(* IEC 61131-3 sources: Lasal/CPU_5344_V01/Class/cmServo, 1 file *)

(* ---- cmServo.st ---- *)
(*!
<Class
	Name               = "cmServo"
	Revision           = "1.0"
	RealtimeTask       = "false"
	CyclicTask         = "true"
	DefCyclictime      = "10 ms"
	BackgroundTask     = "true"
	DefBackground      = "500 ms"
	Sigmatek           = "false"
	OSInterface        = "false"
	HighPriority       = "false"
	Automatic          = "false"
	UpdateMode         = "Prescan"
	SharedCommandTable = "true"
	Objectsize         = "(570,2640)">
	<Channels>
		<Server Name="calcReqSpeed" Visualized="false" Initialize="false" WriteProtected="true" Retentive="false"/>
		<Server Name="csPowerOffServo" Visualized="false" Initialize="false" WriteProtected="false" Retentive="false"/>
		<Server Name="firstPos" Visualized="false" Initialize="false" WriteProtected="false" Retentive="false"/>
		<Server Name="parExtraIFactor" Visualized="true" Initialize="true" DefValue="0" WriteProtected="false" Retentive="File"/>
		<Server Name="parHomeAgain" Visualized="true" Initialize="false" WriteProtected="false" Retentive="false"/>
		<Server Name="parIFactor" Visualized="true" Initialize="true" DefValue="0" WriteProtected="false" Retentive="File"/>
		<Server Name="parInPosBand" Visualized="true" Initialize="true" DefValue="100" WriteProtected="false" Retentive="File" Comment="max difference between act real pos and req pos  (*100)&#13;&#10;in thousands of mm for sts.InPos"/>
		<Server Name="parJogTime" Visualized="true" Initialize="true" DefValue="500" WriteProtected="false" Retentive="File"/>
		<Server Name="parKeepControllerOn" Visualized="true" Initialize="true" WriteProtected="false" Retentive="File"/>
		<Server Name="parLastPieceBand" Visualized="true" Initialize="true" DefValue="1000" WriteProtected="false" Retentive="File"/>
		<Server Name="parManualSpeed" Visualized="true" Initialize="true" DefValue="500" WriteProtected="false" Retentive="File"/>
		<Server Name="parMaxAcc" Visualized="true" Initialize="true" DefValue="10000" WriteProtected="false" Retentive="File"/>
		<Server Name="parMaxDec" Visualized="true" Initialize="true" DefValue="10000" WriteProtected="false" Retentive="File"/>
		<Server Name="parMaxPos" Visualized="true" Initialize="true" DefValue="1500000" WriteProtected="false" Retentive="File"/>
		<Server Name="parMaxSpeed" Visualized="true" Initialize="true" DefValue="10000" WriteProtected="false" Retentive="File"/>
		<Server Name="parMinPos" Visualized="true" Initialize="true" DefValue="0" WriteProtected="false" Retentive="File"/>
		<Server Name="parNoRefSwitch" Visualized="true" Initialize="true" WriteProtected="false" Retentive="File"/>
		<Server Name="parOverrideSimulateServo" Visualized="false" Initialize="false" WriteProtected="false" Retentive="File"/>
		<Server Name="parRefDirPositive" Visualized="true" Initialize="true" DefValue="1" WriteProtected="false" Retentive="File"/>
		<Server Name="parRefPos" Visualized="true" Initialize="true" DefValue="1500000" WriteProtected="false" Retentive="File"/>
		<Server Name="parRefSpeed" Visualized="true" Initialize="true" DefValue="1000" WriteProtected="false" Retentive="File"/>
		<Server Name="parTimeBrakeOff" Visualized="true" Initialize="true" DefValue="200" WriteProtected="false" Retentive="File"/>
		<Server Name="parTimeBrakeOn" Visualized="true" Initialize="true" DefValue="200" WriteProtected="false" Retentive="File"/>
		<Server Name="parTimeControllerOn" Visualized="true" Initialize="true" DefValue="100" WriteProtected="false" Retentive="File"/>
		<Server Name="parTimeOutTime" Visualized="true" Initialize="true" DefValue="120000" WriteProtected="false" Retentive="File"/>
		<Server Name="parWaitInPosTime" Visualized="true" Initialize="true" DefValue="100" WriteProtected="false" Retentive="File"/>
		<Server Name="PendelOn" Visualized="false" Initialize="false" WriteProtected="false" Retentive="false"/>
		<Server Name="reqAcc" Visualized="true" Initialize="false" WriteProtected="false" Retentive="false"/>
		<Server Name="reqDec" Visualized="true" Initialize="false" WriteProtected="false" Retentive="false"/>
		<Server Name="reqPos" Visualized="true" Initialize="false" WriteProtected="false" Retentive="false"/>
		<Server Name="reqSpeed" Visualized="true" Initialize="false" WriteProtected="false" Retentive="false"/>
		<Server Name="secondPos" Visualized="false" Initialize="false" WriteProtected="false" Retentive="false"/>
		<Server Name="stsActRealPos" Visualized="true" Initialize="false" WriteProtected="true" Retentive="false"/>
		<Server Name="stsAllSimuActive" Visualized="false" Initialize="false" WriteProtected="true" Retentive="false"/>
		<Server Name="stsControllerIsOn" Visualized="true" Initialize="false" WriteProtected="true" Retentive="false"/>
		<Server Name="stsInPos" Visualized="true" Initialize="false" WriteProtected="true" Retentive="false"/>
		<Server Name="stsIsHomed" Visualized="true" Initialize="false" WriteProtected="false" Retentive="false"/>
		<Server Name="stsPos" Visualized="true" Initialize="false" WriteProtected="true" Retentive="false"/>
		<Server Name="stsSimRef" Visualized="false" Initialize="false" WriteProtected="true" Retentive="false"/>
		<Server Name="stsSpeed" Visualized="false" Initialize="false" WriteProtected="true" Retentive="false"/>
		<Server Name="stsState" Visualized="true" Initialize="false" WriteProtected="false" Retentive="false"/>
		<Client Name="cntrDistance1" Required="true" Internal="true"/>
		<Client Name="ctrlLiftingCil" Required="false" Internal="false"/>
		<Client Name="iEmergencyStop" Required="false" Internal="false"/>
		<Client Name="iHWReady" Required="true" Internal="false"/>
		<Client Name="iPmSpeed" Required="true" Internal="false" DefValue="1000"/>
		<Client Name="iReleaseMovement" Required="true" Internal="false"/>
		<Client Name="lmcCtrl" Required="true" Internal="false"/>
		<Client Name="oBrake" Required="false" Internal="false"/>
		<Client Name="oIFactor" Required="false" Internal="false"/>
		<Client Name="oResetHW" Required="false" Internal="false"/>
		<Client Name="oSimRefSwitch" Required="false" Internal="false"/>
		<Client Name="sExtraForMinMaxPos" Required="false" Internal="false"/>
		<Client Name="sNoHoming" Required="false" Internal="false" DefValue="0"/>
	</Channels>
	<Separators>
		<Servers>
			<SepChn Position="10"/>
			<SepChn Position="34"/>
			<SepChn Position="40"/>
		</Servers>
	</Separators>
	<RevDoku>
		<Owner Author="JdK"/>
		<Dokumentation Revision="0.3" Date="2020-04-01" Author="TP" Description="add variable speed with ipmSpeed"/>
		<Dokumentation Revision="0.1" Date="2019-10-03" Author="JdK" Description="added control for start homing and merker to home again"/>
		<Dokumentation Revision="0.2" Date="2019-09-24" Author="JdK" Description="added coupling possibillity"/>
	</RevDoku>
	<Network Name="cmServo">
		<!-- List of Components in this network -->
		<Components>
			<Object
				Name       = "_base"
				Class      = "cmBase"
				Position   = "(218,120)"
				Visualized = "true">
				<Channels>
					<Server Name="ClassSvr"/>
					<Server Name="cmdHMI"/>
					<Server Name="ErrorNr"/>
					<Server Name="mode"/>
					<Server Name="state"/>
					<Server Name="stsHMI_RunsAllowed"/>
					<Server Name="stsInAlarm"/>
					<Server Name="stsIsInterlocked"/>
					<Client Name="id"/>
					<Client Name="nwEmOrUnit"/>
				</Channels>
			</Object>
			<Object
				Name           = "cntrDistance1"
				Class          = "cntrDistance"
				Position       = "(300,1110)"
				Visualized     = "true"
				BackgroundTime = "100 ms">
				<Channels>
					<Server Name="actPos"/>
					<Server Name="ClassSvr"/>
					<Server Name="resetSoftCounter"/>
					<Server Name="softCounter"/>
					<Server Name="totalCounter"/>
				</Channels>
			</Object>
		</Components>
		<Comments>
		</Comments>
		<!-- List of Connections in this network -->
		<Connections>
			<Connection Source="this.ClassSvr" Destination="_base.ClassSvr" Vertices="(1036,210),(864,210),"/>
			<Connection Source="this.state" Destination="_base.state" Vertices="(1036,270),(864,270),"/>
			<Connection Source="this.mode" Destination="_base.mode" Vertices="(1036,330),(864,330),"/>
			<Connection Source="this.cmdHMI" Destination="_base.cmdHMI" Vertices="(1036,390),(864,390),"/>
			<Connection Source="this.stsInAlarm" Destination="_base.stsInAlarm" Vertices="(1036,450),(864,510),"/>
			<Connection Source="this.stsIsInterlocked" Destination="_base.stsIsInterlocked" Vertices="(1036,510),(864,570),"/>
			<Connection Source="this.ErrorNr" Destination="_base.ErrorNr" Vertices="(1036,630),(864,690),"/>
			<Connection Source="_base.nwEmOrUnit" Destination="this.nwEmOrUnit" Vertices="(218,210),(38,210),"/>
			<Connection Source="_base.id" Destination="this.id" Vertices="(218,270),(38,270),"/>
			<Connection Source="this.stsHMI_RunsAllowed" Destination="_base.stsHMI_RunsAllowed" Vertices="(1036,570),(864,630),"/>
			<Connection Source="this.cntrDistance1" Destination="cntrDistance1.ClassSvr"/>
		</Connections>
		<!-- Headerfiles -->
		<Options>
		</Options>
	</Network>
</Class>
*)
#pragma using cmBase

cmServo : CLASS
: cmBase
  //Servers:
	stsState 	: SvrCh_servoPos;
	stsIsHomed 	: SvrCh_DINT;
	stsInPos 	: SvrCh_DINT;
	stsControllerIsOn 	: SvrCh_DINT;
	stsPos 	: SvrCh_DINT;
	stsActRealPos 	: SvrCh_DINT;
	stsSpeed 	: SvrCh_DINT;
	stsSimRef 	: SvrCh_DINT;
	stsAllSimuActive 	: SvrCh_DINT;
	csPowerOffServo 	: SvrCh_DINT;
	parMinPos 	: SvrCh_DINT;
	parMaxPos 	: SvrCh_DINT;
	parMaxSpeed 	: SvrCh_DINT;
	parMaxAcc 	: SvrCh_DINT;
	parMaxDec 	: SvrCh_DINT;
	parRefSpeed 	: SvrCh_DINT;
	parRefPos 	: SvrCh_DINT;
	parRefDirPositive 	: SvrCh_DINT;
	parNoRefSwitch 	: SvrCh_DINT;
	parIFactor 	: SvrCh_DINT;
	parExtraIFactor 	: SvrCh_DINT;
	parInPosBand 	: SvrCh_DINT;
	parLastPieceBand 	: SvrCh_DINT;
	parTimeControllerOn 	: SvrCh_UDINT;
	parTimeOutTime 	: SvrCh_UDINT;
	parWaitInPosTime 	: SvrCh_UDINT;
	parTimeBrakeOn 	: SvrCh_UDINT;
	parTimeBrakeOff 	: SvrCh_UDINT;
	parJogTime 	: SvrCh_UDINT;
	parKeepControllerOn 	: SvrCh_DINT;
	parManualSpeed 	: SvrCh_DINT;
	parHomeAgain 	: SvrCh_DINT;
	parOverrideSimulateServo 	: SvrCh_DINT;
	reqPos 	: SvrCh_DINT;
	reqSpeed 	: SvrCh_DINT;
	reqAcc 	: SvrCh_DINT;
	reqDec 	: SvrCh_DINT;
	calcReqSpeed 	: SvrCh_DINT;
	PendelOn 	: SvrCh_DINT;
	firstPos 	: SvrCh_DINT;
	secondPos 	: SvrCh_DINT;
  //Clients:
	lmcCtrl 	: CltChCmd__LMCAxis;
	ctrlLiftingCil 	: CltChCmd_cmCil;
	oIFactor 	: CltCh_DINT;
	oBrake 	: CltCh_DINT;
	oSimRefSwitch 	: CltCh_DINT;
	oResetHW 	: CltCh_DINT;
	iHWReady 	: CltCh_DINT;
	iEmergencyStop 	: CltCh_DINT;
	iReleaseMovement 	: CltCh_DINT;
	iPmSpeed 	: CltCh_DINT;
	sNoHoming 	: CltCh_DINT;
	sExtraForMinMaxPos 	: CltCh_DINT;
	cntrDistance1 	: CltChCmd_cntrDistance;
  //Variables:
		timerTimeOut 	: strTimer;
		timerJog 	: strTimer;
		timerControllerOn 	: strTimer;
		timerWaitInPos 	: strTimer;
		timerBrakeOn 	: strTimer;
		timerBrakeOff 	: strTimer;
		timerSimRef 	: strTimer;
		jogSet 	: DINT;
		tmpRefMode 	: _LMCAXIS_REFMODE;
		tmpAcc 	: DINT;
		tmpDec 	: DINT;
		tmpSpeed 	: DINT;
		tmpOldReqSpeed 	: DINT;
		tmpHomingDone 	: DINT;
		tmpCouplingSpeed 	: DINT;
		tmpCouplingAcc 	: DINT;
		tmpCouplingMaster 	: ^MasterStruct;
		esWasAlreadyActive 	: DINT;
  //Functions:

	FUNCTION VIRTUAL GLOBAL Background
		VAR_INPUT
			EAX 	: UDINT;
		END_VAR
		VAR_OUTPUT
			state (EAX) 	: UDINT;
		END_VAR;

	FUNCTION VIRTUAL execHmiCmd1;

	FUNCTION VIRTUAL execHmiCmd2;

	FUNCTION VIRTUAL execHmiCmd3;

	FUNCTION VIRTUAL resetAlarm;

	FUNCTION VIRTUAL work;

	FUNCTION VIRTUAL execStart;

	FUNCTION VIRTUAL execStop;

	FUNCTION VIRTUAL Init1;

	FUNCTION VIRTUAL preScanOverride;

	FUNCTION VIRTUAL postScanOverride;

	FUNCTION GLOBAL csStartMoveAbs
		VAR_INPUT
			iReqPos 	: DINT;
			iReqSpeed 	: DINT;
		END_VAR;

	FUNCTION VIRTUAL GLOBAL checkInPos
		VAR_INPUT
			checkPos 	: DINT;
		END_VAR
		VAR_OUTPUT
			ok 	: DINT;
		END_VAR;

	FUNCTION GLOBAL giveActualSpeed
		VAR_OUTPUT
			speed 	: DINT;
		END_VAR;

	FUNCTION GLOBAL csStartHoming;

	FUNCTION GLOBAL csStop;

	FUNCTION startMoveAbs
		VAR_INPUT
			iReqPos 	: DINT;
		END_VAR;

	FUNCTION startHoming;

	FUNCTION Pendel;

	FUNCTION GLOBAL csPowerOn;

	FUNCTION GLOBAL csCheckPosFits
		VAR_INPUT
			pos 	: DINT;
		END_VAR
		VAR_OUTPUT
			fits 	: DINT;
		END_VAR;

	FUNCTION GLOBAL csCouple
		VAR_INPUT
			start1Stop0 	: DINT;
			couplingMaxSpeed 	: DINT;
			couplingMaxAcc 	: DINT;
			master 	: ^MasterStruct;
		END_VAR
		VAR_OUTPUT
			done 	: DINT;
		END_VAR;

	FUNCTION GLOBAL csGiveMaster
		VAR_OUTPUT
			master 	: ^MasterStruct;
		END_VAR;

	FUNCTION GLOBAL csPowerOff;

	FUNCTION VIRTUAL GLOBAL parMinPos::Write
		VAR_INPUT
			input (EAX) 	: DINT;
		END_VAR
		VAR_OUTPUT
			result (EAX) 	: DINT;
		END_VAR;

	FUNCTION VIRTUAL GLOBAL parMaxPos::Write
		VAR_INPUT
			input (EAX) 	: DINT;
		END_VAR
		VAR_OUTPUT
			result (EAX) 	: DINT;
		END_VAR;

	FUNCTION VIRTUAL GLOBAL parMaxSpeed::Write
		VAR_INPUT
			input (EAX) 	: DINT;
		END_VAR
		VAR_OUTPUT
			result (EAX) 	: DINT;
		END_VAR;

	FUNCTION VIRTUAL GLOBAL parMaxAcc::Write
		VAR_INPUT
			input (EAX) 	: DINT;
		END_VAR
		VAR_OUTPUT
			result (EAX) 	: DINT;
		END_VAR;

	FUNCTION VIRTUAL GLOBAL reqPos::Write
		VAR_INPUT
			input (EAX) 	: DINT;
		END_VAR
		VAR_OUTPUT
			result (EAX) 	: DINT;
		END_VAR;
  //Tables:
	FUNCTION @STD
		VAR_OUTPUT
			ret_code	: CONFSTATES;
		END_VAR;
	FUNCTION GLOBAL TAB @CT_;
END_CLASS;

#pragma using cntrDistance
#pragma usingLtd _LMCAxis
#pragma usingLtd cmCil

// JdK 3-10-2019: added control sNoHoming = 0 before start homing, also added parHomeAgain, merker for em's to home again if required
// JdK 24-9-2019: added possibility to couple two normally independent servo's
// cmServo created by JdK at 17-5-2019 for library MPS/project 4284
// goal is to control a servo movement icm a LMC object

// HMI start means start movement, HMI stop means stop movement, HMI cmd1: start homing, cmd2: jog positive, cmd3: jog negative

FUNCTION VIRTUAL cmServo::work

  //stsState control
  IF stsState<>seStop & stsState<>seWaitReset & stsState<>seIdle & (pmlCom.sts.isInterlocked=1 | pmlCom.sts.inAlarm=1 | iEmergencyStop=1 | iReleaseMovement=0) THEN
    stsState:=seStop; //if interlock or alarm, stop movement
  END_IF;

  CASE stsState OF

    seStop: //stop movement
      IF lmcCtrl.ActVelocity < 50 & lmcCtrl.ActVelocity > -50 THEN //wait until moving stopped
        stsState:=seWaitReset;
      ELSE
        lmcCtrl.StopMove(Decel:=3*parMaxDec); //sStop movement as fast as possible
      END_IF;

    seWaitReset: //wait until problem is solved
      IF pmlCom.sts.inAlarm=0 & pmlCom.sts.isInterlocked=0 THEN //no problem active, make starting again possible
        stsState:=seIdle;
      END_IF;

    seIdle: //ready for new action

    seWaitStartMoveRef: //wait until controller on/brake released
      IF stsControllerIsOn=1 & timerBrakeOff.done=1 THEN
        stsState:=seStartMoveRef;
      END_IF;

    seStartMoveRef: //give ref command
      tmpRefMode:= _LMCAXIS_REFMODE.NoZImpulse; //we don't use the Z pulse of the encoder
      IF parRefDirPositive THEN //IF DIRECTION IS POSITIVE, TELL IT TO THE CONTROLLER
        tmpRefMode += _LMCAXIS_REFMODE.RefDirection;
      END_IF;
      IF parNoRefSwitch THEN
        tmpRefMode += _LMCAXIS_REFMODE.ESEqualRef; //no refswitch means use endswitch for homing
      END_IF;

      lmcCtrl.Override.Write(input:=1000);//override at max
      lmcCtrl.MoveReference(Mode:=tmpRefMode,
                   Position:=ParRefPos,
                      VRef1:=ParRefSpeed,
                      VRef2:=(ParRefSpeed/5), //reverse direction of homing with 1/5 of normal homing speed
                      Accel:=ParMaxAcc, //use normal acc
             PositionWindow:=ParInPosBand);
      stsState:=seMoveRef;

    seMoveRef: //wait until ref is done
      IF lmcCtrl.AxisStatus.IsReferenced=1 THEN
        tmpHomingDone:= 1;
        parHomeAgain:= 0;
        stsState:=seIdle;
      END_IF;

    seWaitStartMove: //wait until controller on/brake released
      IF stsControllerIsOn=1 & timerBrakeOff.done=1 THEN
        stsState:=seStartMove;
        oIFactor:=parIFactor;
      END_IF;

    seStartMove: //give move command
      IF reqAcc = 0 THEN
        tmpAcc:=ParMaxAcc;//no Acc given, use the max
      ELSE
        tmpAcc:= (reqAcc * parMaxAcc)/1000; //ReqAcc is a percentage of the maximum
      END_IF;
      IF reqDec = 0 THEN
        tmpDec:=parMaxDec;//no Acc given, use the max
      ELSE
        tmpDec:= (reqDec * parMaxDec)/1000; //ReqAcc is a percentage of the maximum
      END_IF;

      IF pmlCom.sts.mode=manual THEN
        tmpSpeed:= parManualSpeed*iPmSpeed/1000; //in manual move with half the speed
      ELSE

        if ReqSpeed = 0 & calcReqSpeed <> 0 then // tp and calcReqSpeed = not null
          reqSpeed:= 1000;
          tmpSpeed:=(1000*iPmSpeed)/1000;
        else
          tmpSpeed := calcReqSpeed;//JdK 5-11-2019: just use given speed, sometimes we want a wagon to hold for some time, so we need speed 0
        end_if;
      END_IF;

      lmcCtrl.Override.Write(input:=tmpSpeed); //required speed is in 1/10%, even as the override, in this way we control the speed
      lmcCtrl.MoveAbsolute(Position:=ReqPos,
                         Speed:=parMaxSpeed,
                         Accel:=tmpAcc,
                         Decel:=tmpDec);
      tmpOldReqSpeed:=calcReqSpeed;
      stsState:=seMove;

    seMove: //wait until movement is nearly done
      IF (lmcCtrl.Destination <> reqPos | tmpOldReqSpeed <> calcReqSpeed ) THEN //start again if req pos or speed changed
        stsState:= seStartMove;
      ELSIF stsInPos=1 then
        stsState := seWaitInPos;
      ELSIF lmcCtrl.InPosition(Mode:=LMCAXIS_POSITIONWINDOW_INT_UNITS, PositionWindow:=parLastPieceBand) =1 THEN
        stsState:= seMoveLastPiece;
      END_IF;

    seMoveLastPiece: //wait until movement is done
      oIFactor:=parExtraIFactor;
      IF ((lmcCtrl.Destination <> reqPos) | tmpOldReqSpeed <> calcReqSpeed  ) THEN //start again if req pos or speed changed
        stsState:= seStartMove;
      ELSIF stsInPos =1 THEN
        stsState:= seWaitInPos;
      END_IF;

    seWaitInPos:
      IF (lmcCtrl.Destination <> reqPos | tmpOldReqSpeed <> calcReqSpeed) THEN //start again if req pos or speed changed
        stsState:= seWaitStartMove;
      ELSIF timerWaitInPos.done=1 THEN
        If stsInPos=1 THEN //action done
          stsState:=seIdle;
        ELSE //start action again
          stsState:=seWaitStartMove;
        END_IF;
      END_IF;

    seWaitStartJogPos:
      IF stsControllerIsOn=1 & timerBrakeOff.done=1 THEN
        stsState:=seStartJogPos;
      END_IF;

    seStartJogPos:
      lmcCtrl.Override.Write(input:=100); //jog at 10% of speed
      lmcCtrl.MoveEndless(Speed:=parMaxSpeed, Accel:=parMaxAcc);
      stsState:=seJogPos;

    seJogPos:
      IF timerJog.done=1 THEN
        stsState:=seStop;
      END_IF;

    seWaitStartJogNeg:
      IF stsControllerIsOn=1 & timerBrakeOff.done=1 THEN
        stsState:=seStartJogNeg;
      END_IF;

    seStartJogNeg:
      lmcCtrl.Override.Write(input:=100); //jog at 10% of speed
      lmcCtrl.MoveEndless(Speed:=parMaxSpeed*-1, Accel:=parMaxAcc);
      stsState:=seJogNeg;

    seJogNeg:
      IF timerJog.done=1 THEN
        stsState:=seStop;
      END_IF;

    seStartCoupling:
      IF stsControllerIsOn=1 & timerBrakeOff.done=1 THEN
        lmcCtrl.CoupleGearRelative(     MaxVel:=parMaxSpeed,
                                        MaxAcc:=parMaxAcc,
                                       pMaster:=tmpCouplingMaster,
                                       GearMul:=1,
                                       GearDiv:=1);//,
                                       //MaxJerk:=);

        stsState:=seWaitCoupling;
      END_IF;

    seWaitCoupling:
      IF lmcCtrl.Control = LOCKED_LMCAXIS THEN
        stsState:=seCoupled;
      END_IF;

    seCoupled:

    seWaitUnCoupling:
      IF lmcCtrl.Control <> LOCKED_LMCAXIS THEN
        stsState:=seIdle;
      ELSE
        lmcCtrl.PowerOff(Mode:=LMCAXIS_IMMEDIATE_STOPP);
      END_IF;

  END_CASE;

  //depending on state, power lmc axis
  IF stsState=seWaitStartMoveRef | stsState=seWaitStartMove | stsState=seWaitStartJogNeg | stsState=seWaitStartJogPos | stsState=seStartCoupling THEN
    lmcCtrl.PowerOn(Mode:=LMCAXIS_MOVE_ANY_WAY);
  END_IF;

  //depending on state and some mor, power off lmc axis
  IF stsControllerIsOn=1 & (stsState=seWaitReset | ((stsState=seIdle | stsState=seWaitInPos) & timerBrakeOn.done=1 & (parKeepControllerOn=0 | csPowerOffServo=1))) THEN //JdK 23-4-2022 make it possible to poweroff servo, in this case (5010) for moving into a toolmagazine, and need one servo to go free
    lmcCtrl.PowerOff(Mode:=LMCAXIS_IMMEDIATE_STOPP);
  END_IF;

END_FUNCTION

FUNCTION GLOBAL cmServo::csStartMoveAbs
	VAR_INPUT
		iReqPos 	: DINT;
		iReqSpeed 	: DINT;
	END_VAR

  IF pmlCom.sts.mode=auto | pmlCom.sts.mode=service THEN
    reqSpeed:=iReqSpeed;
    startMoveAbs(iReqPos:=iReqPos);
  END_IF;

END_FUNCTION

FUNCTION VIRTUAL GLOBAL cmServo::checkInPos
	VAR_INPUT
		checkPos 	: DINT;
	END_VAR
	VAR_OUTPUT
		ok 	: DINT;
	END_VAR

  //real positions should be in 1/1000 of mm, means resolution in LMC is 100
  ok := stsActRealPos<= ((checkPos *lmcCtrl.Resolution)+parInPosBand) & stsActRealPos>= ((checkPos *lmcCtrl.Resolution)-parInPosBand) ;

END_FUNCTION

FUNCTION GLOBAL cmServo::csStartHoming

  //only accept cs commands if in auto/service
  IF (pmlCom.sts.mode=auto | pmlCom.sts.mode=service) & sNoHoming= 0 THEN
    startHoming();
  END_IF;

END_FUNCTION

FUNCTION cmServo::startMoveAbs
	VAR_INPUT
		iReqPos 	: DINT;
	END_VAR

  IF stsState<> seStop & stsState<> seWaitReset THEN //only if not in stop or wait reset
    IF iReqPos <= parMaxPos & iReqPos >= parMinPos THEN
      reqPos:=iReqPos;
      IF stsState<> seWaitStartMove & stsState<> seStartMove & stsState<> seMove & stsState<> seMoveLastPiece & stsState<> seWaitReset THEN
        stsState:=seWaitStartMove;
      END_IF;
    ELSE
      giveAlarm(errorNr:=2);
    END_IF;
  END_IF;

END_FUNCTION

FUNCTION cmServo::startHoming
  //start homing, only if in idle
  IF stsState= seIdle THEN
    stsState:=seWaitStartMoveRef;
  END_IF;

END_FUNCTION

FUNCTION VIRTUAL cmServo::execStart
  //start move from HMI
  startMoveAbs(iReqPos:=reqPos);

END_FUNCTION

FUNCTION VIRTUAL cmServo::execStop
  //execute stop command
  IF stsState<> seStop & stsState<> seWaitReset & (stsState<> seIdle | stsControllerIsOn) THEN //only if not already stopped
    stsState:=seStop;
  END_IF;

END_FUNCTION

FUNCTION VIRTUAL GLOBAL cmServo::Background
	VAR_INPUT
		EAX 	: UDINT;
	END_VAR
	VAR_OUTPUT
		state (EAX) 	: UDINT;
	END_VAR

  lmcCtrl.SWMinPos.Write(input:=parMinPos-sExtraForMinMaxPos); //keep some distance because we don't want alarms if there is some overshoot
  lmcCtrl.SWMaxPos.Write(input:=parMaxPos+sExtraForMinMaxPos);
  sNoHoming:= sNoHoming.Read();

  state:=1;

END_FUNCTION

FUNCTION GLOBAL cmServo::csStop

  IF pmlCom.sts.mode=auto | pmlCom.sts.mode=service THEN
    execStop();
  END_IF;

END_FUNCTION

FUNCTION VIRTUAL cmServo::resetAlarm

  _Alarm.AlarmActief.Write(input:=0);
  _Alarm.ErrorNr.Write(input:=0);
  IF (stsState= seWaitReset | stsState=seIdle) & lmcCtrl.AxisError<>0 THEN
    oResetHW.Write(input:=1);
    lmcCtrl.QuitError();
  END_IF;

END_FUNCTION

FUNCTION VIRTUAL GLOBAL cmServo::reqPos::Write
	VAR_INPUT
		input (EAX) 	: DINT;
	END_VAR
	VAR_OUTPUT
		result (EAX) 	: DINT;
	END_VAR

  IF pmlCom.sts.mode= manual | pmlCom.sts.mode= service THEN //only take write of new pos if in manual
	  reqPos := input;
  END_IF;

	result := reqPos;

END_FUNCTION

FUNCTION VIRTUAL cmServo::execHmiCmd1
//hmi start home
  startHoming();

END_FUNCTION

FUNCTION VIRTUAL cmServo::execHmiCmd2
//hmi start jog pos
  IF stsState<> seStop & stsState<> seWaitReset & stsState<> seWaitStartJogPos & stsState<> seStartJogPos & stsState<> seJogPos THEN
    stsState:=seWaitStartJogPos;
  END_IF;
  jogSet:=1; //to set timer again

END_FUNCTION

FUNCTION VIRTUAL cmServo::execHmiCmd3
//hmi start jog pos
  IF stsState<> seStop & stsState<> seWaitReset & stsState<> seWaitStartJogNeg & stsState<> seStartJogNeg & stsState<> seJogNeg THEN
    stsState:=seWaitStartJogNeg;
  END_IF;
  jogSet:=1; //to set timer again

END_FUNCTION

FUNCTION cmServo::Pendel
  //method is only called if pendel is active, is meant to see how movement goes and to tune PID params
  IF stsState= seIdle THEN //in idle so go to next pos
    IF reqPos=firstPos THEN
      startMoveAbs(iReqPos:=secondPos);
    ELSE
      startMoveAbs(iReqPos:=firstPos);
    END_IF;
  END_IF;

END_FUNCTION

FUNCTION VIRTUAL cmServo::Init1

  IF initDone=0 THEN
    //write minpos, maxpos, speed and acc
    sExtraForMinMaxPos:=sExtraForMinMaxPos.Read(); //make extra space for min/max pos optional changeble
    IF sExtraForMinMaxPos=0 THEN
      sExtraForMinMaxPos:=20;
    END_IF;

    lmcCtrl.SWMinPos.Write(input:=parMinPos-sExtraForMinMaxPos); //keep some distance because we don't want alarms if there is some overshoot
    lmcCtrl.SWMaxPos.Write(input:=parMaxPos+sExtraForMinMaxPos);
    lmcCtrl.VMax.Write(input:=parMaxSpeed);
    lmcCtrl.AMax.Write(input:=parMaxAcc);
    //lmcCtrl.Resolution.Write(input:=1000);
    IF parManualSpeed=0 THEN
      parManualSpeed:=100; //set speed at 10%
    END_IF;
    initDone:=1;

  END_IF;

  tmpHomingDone:= 0;

END_FUNCTION

FUNCTION GLOBAL cmServo::giveActualSpeed
	VAR_OUTPUT
		speed 	: DINT;
	END_VAR
  //method to give actual speed in % of maximum
  IF parMaxSpeed <> 0 THEN
    speed:=(lmcCtrl.ActVelocity*1000)/parMaxSpeed;
  ELSE
    speed:=0;
  END_IF;

END_FUNCTION

FUNCTION VIRTUAL GLOBAL cmServo::parMinPos::Write
	VAR_INPUT
		input (EAX) 	: DINT;
	END_VAR
	VAR_OUTPUT
		result (EAX) 	: DINT;
	END_VAR

	parMinPos := input;
  lmcCtrl.SWMinPos.Write(input:=parMinPos-sExtraForMinMaxPos); //keep some distance because we don't want alarms if there is some overshoot
	result := parMinPos;

END_FUNCTION

FUNCTION VIRTUAL GLOBAL cmServo::parMaxPos::Write
	VAR_INPUT
		input (EAX) 	: DINT;
	END_VAR
	VAR_OUTPUT
		result (EAX) 	: DINT;
	END_VAR

	parMaxPos := input;
  lmcCtrl.SWMaxPos.Write(input:=parMaxPos+sExtraForMinMaxPos);
	result := parMaxPos;

END_FUNCTION

FUNCTION VIRTUAL GLOBAL cmServo::parMaxSpeed::Write
	VAR_INPUT
		input (EAX) 	: DINT;
	END_VAR
	VAR_OUTPUT
		result (EAX) 	: DINT;
	END_VAR

	parMaxSpeed := input;
  lmcCtrl.VMax.Write(input:=parMaxSpeed);
	result := parMaxSpeed;

END_FUNCTION

FUNCTION VIRTUAL GLOBAL cmServo::parMaxAcc::Write
	VAR_INPUT
		input (EAX) 	: DINT;
	END_VAR
	VAR_OUTPUT
		result (EAX) 	: DINT;
	END_VAR

	parMaxAcc := input;
  lmcCtrl.AMax.Write(input:=parMaxAcc);
	result := parMaxAcc;

END_FUNCTION

FUNCTION VIRTUAL cmServo::preScanOverride

  //if servo hardware is frequency controller or something, we may have a ready signal
  iHWReady:=iHWReady.Read();
  iEmergencyStop:=iEmergencyStop.Read();
  IF stsState<> seIdle & stsState<> seWaitReset & stsState<> seStop THEN
    iReleaseMovement:=iReleaseMovement.Read(); //if there is no release, alarm is given in release class
  END_IF;

  //get position in calculation value of lmc, normally this is in 1/1000mm
  stsActRealPos:=lmcCtrl.ReadPosition(Mode:=LMCAXIS_ACTPOS_INTUNIT);

  //calculate in pos state, reqpos is in 1/10 mm, act real pos in 1/1000
  stsInPos:= ABS(stsActRealPos-(reqPos*lmcCtrl.Resolution))< parInPosBand;

  IF stsIsHomed=0 THEN //don't give real value if we are not homed yet
    stsPos:=NOREFVALUE;
  ELSIF stsInPos=1 THEN
    stsPos:=reqPos;
  ELSE
    stsPos:=(stsActRealPos)/lmcCtrl.Resolution; //JdK 23-3-2022 get real resolution  100; //go from 1/1000ste to 1/10
  END_IF;
  stsSpeed:=lmcCtrl.ActVelocity.Read();

  //call timers
  timerTimeOut:=runTimer(Active:=stsState=seMove, iMem:=timerTimeOut, TimerTime:=parTimeOutTime, Pause:=tmpSpeed = 0);//tp 25-09-2020 pause timer when speed is nul
  timerJog:=runTimer(Active:=(stsState=seJogNeg|stsState=seJogPos)&jogSet=0, iMem:=timerJog, TimerTime:=parJogTime, Pause:=0);
  jogSet:=0; //set it to zero every cycle, if button is pressed, it is ma de 1
  timerControllerOn:=runTimer(Active:=lmcCtrl.AxisStatus.PowerOn, iMem:=timerControllerOn, TimerTime:=parTimeControllerOn, Pause:=0);
  timerWaitInPos:=runTimer(Active:=stsState=seWaitInPos, iMem:=timerWaitInPos, TimerTime:=parWaitInPosTime, Pause:=0);
  timerBrakeOn:=runTimer(Active:=oBrake=1, iMem:=timerBrakeOn, TimerTime:=parTimeBrakeOn, Pause:=0);
  timerBrakeOff:=runTimer(Active:=oBrake=0, iMem:=timerBrakeOff, TimerTime:=parTimeBrakeOff, Pause:=0);
  timerSimRef:=runTimer(Active:=stsState=seMoveRef, iMem:=timerSimRef, TimerTime:=10, Pause:=0);

  //homed status
  stsIsHomed:=(lmcCtrl.AxisStatus.IsReferenced);//test JdK 19-7-2019 & (tmpHomingDone=1 | pmlCom.cmd.simulation= allSimu)); //only if homing is started at least once, or no homing required

  //controller on status
  stsControllerIsOn:=timerControllerOn.done;

  //calculate calc req speed
  iPmSpeed:=iPmSpeed.Read();
  calcReqSpeed:= (reqSpeed * iPmSpeed)/1000;

  IF stsControllerIsOn=0 & (lmcCtrl.AxisError.HwMinError=1 | lmcCtrl.AxisError.HwMaxError= 1) THEN //JdK 22-09-2021, don't give alarm after startup, because servo can go down on endswitch
    esWasAlreadyActive:=1;
  ELSIF lmcCtrl.AxisError.HwMinError=0 & lmcCtrl.AxisError.HwMaxError= 0 THEN
    esWasAlreadyActive:= 0;
  END_IF;

  //set alarms
  IF timerTimeOut.done THEN
    giveAlarm(errorNr:=1);
  END_IF;
  //nr 2 is given if reqpos is out of reach
  IF iHWReady= 0 & stsState<>seWaitReset & stsState<>seIdle & stsState<>seStop & pmlCom.cmd.simulation<>allSimu THEN
    giveAlarm(errorNr:=3);
  END_IF;
  IF lmcCtrl.AxisError<>0 & stsState<>seWaitReset & stsState<>seIdle & stsState<>seStop & (esWasAlreadyActive=0 | (lmcCtrl.AxisError.HwMinError=0 & lmcCtrl.AxisError.HwMaxError= 0)) THEN //error in drive, and not stopped
    IF lmcCtrl.AxisError.HwError THEN
      giveAlarm(errorNr:=4);
    ELSIF lmcCtrl.AxisError.SwMinError THEN
      IF stsState=seMove & reqPos < stsPos THEN //only if moving negative
        giveAlarm(errorNr:=5);
      END_IF;
    ELSIF lmcCtrl.AxisError.SwMaxError THEN
      IF stsState=seMove & reqPos > stsPos THEN //only if moving positive
        giveAlarm(errorNr:=6);
      END_IF;
    ELSIF lmcCtrl.AxisError.HwMinError THEN
      IF stsState=seMove & reqPos < stsPos THEN //only if moving negative
        giveAlarm(errorNr:=7);
      END_IF;
    ELSIF lmcCtrl.AxisError.HwMaxError THEN
      IF stsState=seMove & reqPos > stsPos THEN //only if moving positive
        giveAlarm(errorNr:=8);
      END_IF;
    ELSIF lmcCtrl.AxisError.ReferenceError THEN
      giveAlarm(errorNr:=9);
    ELSIF lmcCtrl.AxisError.ContouringError THEN
      giveAlarm(errorNr:=10);
    ELSE
      giveAlarm(errorNr:=11); //general alarm, one of the other alarms is active in the controller
    END_IF;
  END_IF;
  IF iEmergencyStop=1 & stsState<>seWaitReset & stsState<>seIdle & stsState<>seStop THEN
    giveAlarm(errorNr:=12);
  END_IF;

  IF PendelOn=1 & stsIsHomed=1 THEN
    Pendel();
  END_IF;

END_FUNCTION

FUNCTION VIRTUAL cmServo::postScanOverride

  oBrake:= stsState=seWaitReset | ((stsState=seIdle | stsState=seWaitInPos) & ((parKeepControllerOn=0 | csPowerOffServo=1) | stsControllerIsOn=0)); //brake on if reset, or if in idle/wait and not keep controller on, or controller is of
  oBrake.Write(input:=oBrake);

  oIFactor.Write(input:=oIFactor);
  stsSimRef:=(pmlCom.cmd.simulation=allSimu | parOverrideSimulateServo) & stsState=seMoveRef & timerSimRef.done=0;
  stsAllSimuActive:= pmlCom.cmd.simulation= allSimu | parOverrideSimulateServo;

  IF (pmlCom.cmd.simulation=allSimu | parOverrideSimulateServo) & lmcCtrl.SimulateMode<>1 THEN //JdK 7-4-2022: make it possible to test with one or more servo's in simulate mode
    lmcCtrl.SimulateMode.Write(input:=1);
  ELSIF (pmlCom.cmd.simulation<>allSimu & parOverrideSimulateServo=0) & lmcCtrl.SimulateMode<>0 THEN
    lmcCtrl.SimulateMode.Write(input:=0);
  END_IF;

  cntrDistance1.actPos:= stsActRealPos/100; //for counting distance

END_FUNCTION

FUNCTION GLOBAL cmServo::csPowerOn

  //only accept cs commands if in auto/service
  IF (pmlCom.sts.mode=auto | pmlCom.sts.mode=service) & stsControllerIsOn=0 THEN
    lmcCtrl.PowerOn(Mode:=LMCAXIS_MOVE_ANY_WAY);
  END_IF;

END_FUNCTION

FUNCTION GLOBAL cmServo::csCheckPosFits
	VAR_INPUT
		pos 	: DINT;
	END_VAR
	VAR_OUTPUT
		fits 	: DINT;
	END_VAR

  IF pos <= parMaxPos & pos >= parMinPos THEN
    fits:=1;
  ELSE
    fits:=0;
  END_IF;

END_FUNCTION

FUNCTION GLOBAL cmServo::csCouple
	VAR_INPUT
		start1Stop0 	: DINT;
		couplingMaxSpeed 	: DINT;
		couplingMaxAcc 	: DINT;
		master 	: ^MasterStruct;
	END_VAR
	VAR_OUTPUT
		done 	: DINT;
	END_VAR

  done:=0;
  //only accept cs commands if in auto/service
  IF (pmlCom.sts.mode=auto | pmlCom.sts.mode=service) THEN
    IF start1Stop0= 1 THEN //means start coupling
      IF stsState= seIdle THEN
        tmpCouplingSpeed:=couplingMaxSpeed;
        tmpCouplingAcc:=couplingMaxAcc;
        tmpCouplingMaster:=master;
        stsState:= seStartCoupling;
      ELSIF stsState= seCoupled THEN
        done:= 1;
      END_IF;
    ELSE
      IF stsState= seCoupled THEN
        stsState:= seWaitUnCoupling;
      ELSIF stsState= seIdle THEN
        done:= 1;
      END_IF;
    END_IF;
  ELSE
    done:= -1; //failure
  END_IF;

END_FUNCTION

FUNCTION GLOBAL cmServo::csGiveMaster
	VAR_OUTPUT
		master 	: ^MasterStruct;
	END_VAR

  master:=lmcCtrl.ReadMasterInfo(usDelay:=0);

END_FUNCTION

FUNCTION GLOBAL cmServo::csPowerOff

  lmcCtrl.PowerOff(Mode:=LMCAXIS_IMMEDIATE_STOPP);

END_FUNCTION
